Fanuc TP program (LS listing): test_ls_pns.ls

/PROG  test_ls_pns
/ATTR
OWNER		= MNEDITOR;
COMMENT		= "";
PROG_SIZE	= 187;
CREATE		= DATE 20-06-16  TIME 22:32:48;
MODIFIED	= DATE 20-06-16  TIME 22:33:12;
FILE_NAME	= ;
VERSION		= 0;
LINE_COUNT	= 1;
MEMORY_SIZE	= 563;
PROTECT		= READ_WRITE;
TCD:  STACK_SIZE	= 0,
      TASK_PRIORITY	= 50,
      TIME_SLICE	= 0,
      BUSY_LAMP_OFF	= 0,
      ABORT_REQUEST	= 0,
      PAUSE_REQUEST	= 0;
DEFAULT_GROUP	= *,*,*,*,*;
CONTROL_CODE	= 00000000 00000000;
/APPL

AUTO_SINGULARITY_HEADER;
  ENABLE_SINGULARITY_AVOIDANCE   : TRUE;
/MN
   1:  CALL PNS2SR(1) ;
/POS
/END
